// TIA Portal project "Project2" (V17)
// physical plc demo

(* hardware
DEVICE "S7-1500/ET200MP station_1"  S7-1500 station
   slot 0: "Rail_0"  Rack  6ES7 590-1***0-0AA0
   slot 1: "PLC_1"  CPU 1511-1 PN  6ES7 511-1AK02-0AB0  V2.9
      slot 3: "CPU display_1"  6ES7591-1AA00-0AA0
      slot 32768: "PROFINET interface_1"  X1
         slot 32769: "Port_1"  X1 P1
         slot 32770: "Port_2"  X1 P2
      slot 34817: "Virtual CP interface port_1"  Virtual CP interface port  Virtual CP interface port
DEVICE "HMI_1"  TP700 Comfort
   slot 0: "HMI_1"  TP700 Comfort  6AV2 124-0GC01-0AX0  17.0.0.0
   slot 1: "HMI_RT_1"  TP700 Comfort  6AV2 124-0GC01-0AX0  17.0.0.0
   slot 5: "HMI_1.IE_CP_1"  PROFINET Interface  17.0.0.0
      slot 1: "PROFINET Interface_1"  PROFINET Interface
         slot 1: "Port_1"  Port
         slot 2: "Port_2"  Port
   slot 7: "HMI_1.MPI/DP_CP_1"  MPI/DP Interface  17.0.0.0
DEVICE "ET 200SP station_1"  ET 200SP-Station
   slot 0: "RIO"  IM 155-6 PN/2 HF  6ES7 155-6AU01-0CN0  V4.2
   slot 0: "Rack_0"  Rack  6ES5 710-8MAx1
   slot 1: "DI 16x24VDC ST_1"  DI 16x24VDC ST  6ES7 131-6BH01-0BA0  V0.0
      slot 1: "DI 16x24VDC ST_1"  DI 16x24VDC ST
   slot 2: "DQ 16x24VDC/0.5A ST_1"  DQ 16x24VDC/0.5A ST  6ES7 132-6BH01-0BA0  V0.0
      slot 1: "DQ 16x24VDC/0.5A ST_1"  DQ 16x24VDC/0.5A ST
   slot 3: "AI 8xI 2-,4-wire BA_1"  AI 8xI 2-,4-wire BA  6ES7 134-6GF00-0AA1  V1.0
      slot 1: "AI 8xI 2-,4-wire BA_1"  AI 8xI 2-,4-wire BA
   slot 4: "AQ 4xU/I ST_1"  AQ 4xU/I ST  6ES7 135-6HD00-0BA1  V1.1
      slot 1: "AQ 4xU/I ST_1"  AQ 4xU/I ST
   slot 5: "Server module_1"  Server module  6ES7 193-6PA00-0AA0  V1.1
      slot 1: "Server module_1"  Server module
   slot 127: "BA 2xRJ45"  BA 2xRJ45  6ES7 193-6AR00-0AA0  V0.0
      slot 1: "Port_1"  X1 P1 R  6ES7 193-6AR00-0AA0  V0.0
      slot 2: "Port_2"  X1 P2 R  6ES7 193-6AR00-0AA0  V0.0
*)

// ===== PLC "PLC_1"  CPU 1511-1 PN =====

VAR_GLOBAL   // PLC tag table "Default tag table"
   "System_Byte" AT %MB1 : Byte;
   "FirstScan" AT %M1.0 : Bool;
   "DiagStatusUpdate" AT %M1.1 : Bool;
   "AlwaysTRUE" AT %M1.2 : Bool;
   "AlwaysFALSE" AT %M1.3 : Bool;
   "Clock_Byte" AT %MB0 : Byte;
   "Clock_10Hz" AT %M0.0 : Bool;
   "Clock_5Hz" AT %M0.1 : Bool;
   "Clock_2.5Hz" AT %M0.2 : Bool;
   "Clock_2Hz" AT %M0.3 : Bool;
   "Clock_1.25Hz" AT %M0.4 : Bool;
   "Clock_1Hz" AT %M0.5 : Bool;
   "Clock_0.625Hz" AT %M0.6 : Bool;
   "Clock_0.5Hz" AT %M0.7 : Bool;
   "Motor_Cikis" AT %QW2 : Int;
   "Motor_Ariza" AT %I0.0 : Bool;
END_VAR

DATA_BLOCK "Program_parameters_DB"   // DB1
{ S7_Optimized_Access := 'TRUE' }
VERSION : 0.1
   VAR
      QMotor1_Start : Bool;
      QMotor2_Start : Bool;
      QMotor3_Start : Bool;
      IMotor1_Fault : Bool;
      IMotor2_Fault : Bool;
      IMotor3_Fault : Bool;
      AQMotor1_Freq : Int;
      AQMotor2_Freq : Int;
      AQMotor3_Freq : Int;
   END_VAR
BEGIN
END_DATA_BLOCK

DATA_BLOCK "HMI_parameters_DB"   // DB2
{ S7_Optimized_Access := 'TRUE' }
VERSION : 0.1
   VAR
      HMI_Mode_Auto : Bool;
      HMI_M1_Manual_Start : Bool;
      HMI_M2_Manual_Start : Bool;
      HMI_M3_Manual_Start : Bool;
      HMI_M1_Manual_Speed : Real;
      HMI_M2_Manual_Speed : Real;
      HMI_M3_Manual_Speed : Real;
      HMI_M1_Running : Bool;
      HMI_M2_Running : Bool;
      HMI_M3_Running : Bool;
      HMI_M1_Fault : Bool;
      HMI_M2_Fault : Bool;
      HMI_M3_Fault : Bool;
   END_VAR
BEGIN
END_DATA_BLOCK

DATA_BLOCK "FB_Motor3_Sürücü_DB"   // DB3
{ S7_Optimized_Access := 'TRUE' }
VERSION : 0.1
// stored: InstanceOfName FB_Motor_Sürücü
"FB_Motor_Sürücü"
BEGIN
END_DATA_BLOCK

DATA_BLOCK "Data_block_1"   // DB4
{ S7_Optimized_Access := 'TRUE' }
VERSION : 0.1
   VAR
      man : Bool;
      Alarm : Int;
   END_VAR
BEGIN
END_DATA_BLOCK

DATA_BLOCK "FB_Motor1_Sürücü_DB"   // DB6
{ S7_Optimized_Access := 'TRUE' }
VERSION : 0.1
// stored: InstanceOfName FB_Motor_Sürücü
"FB_Motor_Sürücü"
BEGIN
END_DATA_BLOCK

DATA_BLOCK "FB_Motor2_Sürücü_DB"   // DB7
{ S7_Optimized_Access := 'TRUE' }
VERSION : 0.1
// stored: InstanceOfName FB_Motor_Sürücü
"FB_Motor_Sürücü"
BEGIN
END_DATA_BLOCK

FUNCTION_BLOCK "FB_Motor_Sürücü"   // FB1, LAD
{ S7_Optimized_Access := 'TRUE' }
VERSION : 0.1
   VAR_INPUT
      Enable : Bool;
      Mo_Auto : Bool;
      Man_Start : Bool;
      Man_Speed_Hz : Real;
      Driver_Fault : Bool;
   END_VAR
   VAR_OUTPUT
      Start_Out : Bool;
      Analog_Out : Int;
      Running : Bool;
      Alarm : Bool;
   END_VAR
   VAR_TEMP
      Target_Hz : Real;
      Norm_Val : Real;
   END_VAR
BEGIN

REGION Network 1
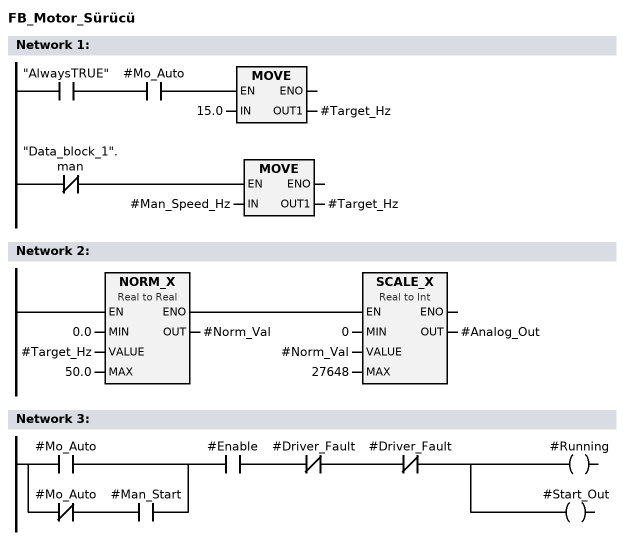
   RUNG wire#powerrail
      Contact( "AlwaysTRUE" )
      Contact( #Mo_Auto )
      Move(in := 15.0, out1 => #Target_Hz)
   END_RUNG
   RUNG wire#powerrail
      I_Contact( "Data_block_1".man )
      Move(in := #Man_Speed_Hz, out1 => #Target_Hz)
   END_RUNG
   // the same network as SCL:
   IF "AlwaysTRUE" AND #Mo_Auto THEN #Target_Hz := 15.0; END_IF;
   IF NOT "Data_block_1".man THEN #Target_Hz := #Man_Speed_Hz; END_IF;
END_REGION

REGION Network 2
   RUNG wire#powerrail
      { S7_Templates := "[SrcType := Real, DestType := Real]" } Normalize(min := 0.0, value := #Target_Hz, max := 50.0, out => #Norm_Val)
      { S7_Templates := "[SrcType := Real, DestType := Int]" } Scale(min := 0, value := #Norm_Val, max := 27648, out => #Analog_Out)
   END_RUNG
   // the same network as SCL:
   #Norm_Val := NORM_X(MIN := 0.0, VALUE := #Target_Hz, MAX := 50.0);
   #Analog_Out := SCALE_X(MIN := 0, VALUE := #Norm_Val, MAX := 27648);
END_REGION

REGION Network 3
   RUNG wire#powerrail
      Contact( #Mo_Auto )
      wire#w1
      Contact( #Enable )
      I_Contact( #Driver_Fault )
      I_Contact( #Driver_Fault )
      wire#w2
      Coil( #Running )
   END_RUNG
   RUNG wire#powerrail
      I_Contact( #Mo_Auto )
      Contact( #Man_Start )
   END_RUNG wire#w1
   RUNG wire#w2
      Coil( #Start_Out )
   END_RUNG
   // the same network as SCL:
   #Running := (#Mo_Auto OR (NOT #Mo_Auto AND #Man_Start)) AND #Enable AND NOT #Driver_Fault AND NOT #Driver_Fault;
   #Start_Out := #Running;
END_REGION
END_FUNCTION_BLOCK

FUNCTION "FC_Example" : Void   // FC1, LAD
{ S7_Optimized_Access := 'TRUE' }
VERSION : 0.1
BEGIN
END_FUNCTION

ORGANIZATION_BLOCK "Main"   // OB1, LAD, ProgramCycle
TITLE = "Main Program Sweep (Cycle)"
{ S7_Optimized_Access := 'TRUE' }
VERSION : 0.1
   VAR_INPUT
      Initial_Call : Bool;   // Initial call of this OB
      Remanence : Bool;   // =True, if remanent data are available
   END_VAR
BEGIN

REGION Network 1
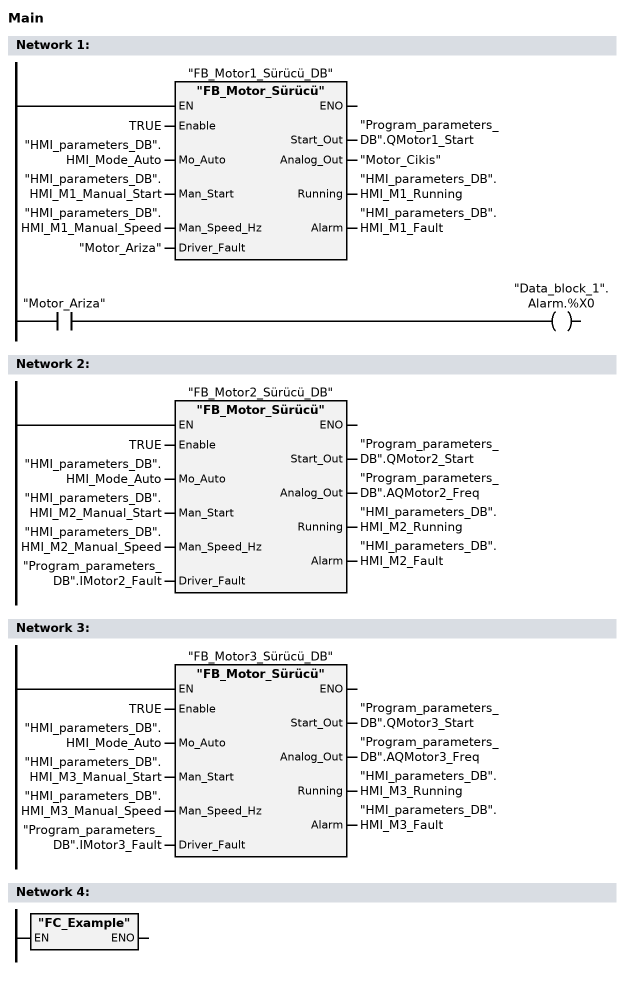
   RUNG wire#powerrail
      "FB_Motor1_Sürücü_DB"(Enable := TRUE, Mo_Auto := "HMI_parameters_DB".HMI_Mode_Auto, Man_Start := "HMI_parameters_DB".HMI_M1_Manual_Start, Man_Speed_Hz := "HMI_parameters_DB".HMI_M1_Manual_Speed, Driver_Fault := "Motor_Ariza", Start_Out => "Program_parameters_DB".QMotor1_Start, Analog_Out => "Motor_Cikis", Running => "HMI_parameters_DB".HMI_M1_Running, Alarm => "HMI_parameters_DB".HMI_M1_Fault)
   END_RUNG
   RUNG wire#powerrail
      Contact( "Motor_Ariza" )
      Coil( "Data_block_1".Alarm.%X0 )
   END_RUNG
   // the same network as SCL:
   "FB_Motor1_Sürücü_DB"(Enable := TRUE,   // "FB_Motor_Sürücü"
                         Mo_Auto := "HMI_parameters_DB".HMI_Mode_Auto,
                         Man_Start := "HMI_parameters_DB".HMI_M1_Manual_Start,
                         Man_Speed_Hz := "HMI_parameters_DB".HMI_M1_Manual_Speed,
                         Driver_Fault := "Motor_Ariza",
                         Start_Out => "Program_parameters_DB".QMotor1_Start,
                         Analog_Out => "Motor_Cikis",
                         Running => "HMI_parameters_DB".HMI_M1_Running,
                         Alarm => "HMI_parameters_DB".HMI_M1_Fault);
   "Data_block_1".Alarm.%X0 := "Motor_Ariza";
END_REGION

REGION Network 2
   RUNG wire#powerrail
      "FB_Motor2_Sürücü_DB"(Enable := TRUE, Mo_Auto := "HMI_parameters_DB".HMI_Mode_Auto, Man_Start := "HMI_parameters_DB".HMI_M2_Manual_Start, Man_Speed_Hz := "HMI_parameters_DB".HMI_M2_Manual_Speed, Driver_Fault := "Program_parameters_DB".IMotor2_Fault, Start_Out => "Program_parameters_DB".QMotor2_Start, Analog_Out => "Program_parameters_DB".AQMotor2_Freq, Running => "HMI_parameters_DB".HMI_M2_Running, Alarm => "HMI_parameters_DB".HMI_M2_Fault)
   END_RUNG
   // the same network as SCL:
   "FB_Motor2_Sürücü_DB"(Enable := TRUE,   // "FB_Motor_Sürücü"
                         Mo_Auto := "HMI_parameters_DB".HMI_Mode_Auto,
                         Man_Start := "HMI_parameters_DB".HMI_M2_Manual_Start,
                         Man_Speed_Hz := "HMI_parameters_DB".HMI_M2_Manual_Speed,
                         Driver_Fault := "Program_parameters_DB".IMotor2_Fault,
                         Start_Out => "Program_parameters_DB".QMotor2_Start,
                         Analog_Out => "Program_parameters_DB".AQMotor2_Freq,
                         Running => "HMI_parameters_DB".HMI_M2_Running,
                         Alarm => "HMI_parameters_DB".HMI_M2_Fault);
END_REGION

REGION Network 3
   RUNG wire#powerrail
      "FB_Motor3_Sürücü_DB"(Enable := TRUE, Mo_Auto := "HMI_parameters_DB".HMI_Mode_Auto, Man_Start := "HMI_parameters_DB".HMI_M3_Manual_Start, Man_Speed_Hz := "HMI_parameters_DB".HMI_M3_Manual_Speed, Driver_Fault := "Program_parameters_DB".IMotor3_Fault, Start_Out => "Program_parameters_DB".QMotor3_Start, Analog_Out => "Program_parameters_DB".AQMotor3_Freq, Running => "HMI_parameters_DB".HMI_M3_Running, Alarm => "HMI_parameters_DB".HMI_M3_Fault)
   END_RUNG
   // the same network as SCL:
   "FB_Motor3_Sürücü_DB"(Enable := TRUE,   // "FB_Motor_Sürücü"
                         Mo_Auto := "HMI_parameters_DB".HMI_Mode_Auto,
                         Man_Start := "HMI_parameters_DB".HMI_M3_Manual_Start,
                         Man_Speed_Hz := "HMI_parameters_DB".HMI_M3_Manual_Speed,
                         Driver_Fault := "Program_parameters_DB".IMotor3_Fault,
                         Start_Out => "Program_parameters_DB".QMotor3_Start,
                         Analog_Out => "Program_parameters_DB".AQMotor3_Freq,
                         Running => "HMI_parameters_DB".HMI_M3_Running,
                         Alarm => "HMI_parameters_DB".HMI_M3_Fault);
END_REGION

REGION Network 4
   RUNG wire#powerrail
      "FC_Example"()
   END_RUNG
   // the same network as SCL:
   "FC_Example"();
END_REGION
END_ORGANIZATION_BLOCK

(* ===== HMI "HMI_RT_1" =====
system functions are stored by id; their names below are inferred from use
connection "HMI_Connection_1": ETHERNET, S7_1500_OMS

HMI tags "Default tag table"
   "Tag_ScreenNumber" : UInt, internal
   "Data_block_1_Alarm" : Int = PLC Data_block_1.Alarm, 1 s
   "HMI_parameters_DB_HMI_Mode_Auto" : Bool = PLC HMI_parameters_DB.HMI_Mode_Auto, 1 s
   "HMI_parameters_DB_HMI_M1_Running" : Bool = PLC HMI_parameters_DB.HMI_M1_Running, 1 s
   "HMI_parameters_DB_HMI_M2_Running" : Bool = PLC HMI_parameters_DB.HMI_M2_Running, 1 s
   "HMI_parameters_DB_HMI_M3_Running" : Bool = PLC HMI_parameters_DB.HMI_M3_Running, 1 s
   "HMI_parameters_DB_HMI_M1_Manual_Start" : Bool = PLC HMI_parameters_DB.HMI_M1_Manual_Start, 1 s
   "HMI_parameters_DB_HMI_M2_Manual_Start" : Bool = PLC HMI_parameters_DB.HMI_M2_Manual_Start, 1 s
   "HMI_parameters_DB_HMI_M3_Manual_Start" : Bool = PLC HMI_parameters_DB.HMI_M3_Manual_Start, 1 s
   "HMI_parameters_DB_HMI_M1_Manual_Speed" : Real = PLC HMI_parameters_DB.HMI_M1_Manual_Speed, 1 s
   "HMI_parameters_DB_HMI_M2_Manual_Speed" : Real = PLC HMI_parameters_DB.HMI_M2_Manual_Speed, 1 s
   "HMI_parameters_DB_HMI_M3_Manual_Speed" : Real = PLC HMI_parameters_DB.HMI_M3_Manual_Speed, 1 s
   "HMI_parameters_DB_HMI_M1_Fault" : Bool = PLC HMI_parameters_DB.HMI_M1_Fault, 1 s
   "HMI_parameters_DB_HMI_M2_Fault" : Bool = PLC HMI_parameters_DB.HMI_M2_Fault, 1 s
   "HMI_parameters_DB_HMI_M3_Fault" : Bool = PLC HMI_parameters_DB.HMI_M3_Fault, 1 s

discrete alarms
   1: 'First Motor Driver Fault!', class Errors, trigger "HMI_parameters_DB_HMI_M1_Fault" bit 0

Template "Template_1" 800x420
   Button "Exit" at 720,360 size 78x58; TextOff 'Exit'; PictureOff "ExitRuntime_TP700_Comfort_TR"; PictureOn "ExitRuntime_TP700_Comfort_TR"
      on Release: StopRuntime(0)
   Button "Template_Button" at 640,360 size 78x58; TextOff 'Text'
   Button "Template_Button_1" at 560,360 size 78x58; TextOff 'Text'
   Button "Template_Button_2" at 480,360 size 78x58; TextOff 'Text'
   Button "Template_Button_3" at 400,360 size 78x58; TextOff 'Text'
   Button "Template_Button_4" at 321,360 size 78x58; TextOff 'Text'
   Button "Template_Button_5" at 241,360 size 78x58; TextOff 'Text'
   Button "Template_Button_6" at 161,360 size 78x58; TextOff 'Text'
   Button "Alarms" at 81,360 size 78x58; TextOff 'Alarms'; PictureOff "AlarmDisplay_TP700_Comfort_TR"; PictureOn "AlarmDisplay_TP700_Comfort_TR"
      on Release: function_ef3f5d25("Alarm window_Unacknowledged", -1)
   Button "Start screen" at 1,360 size 78x58; TextOff 'Start screen'; PictureOff "NavigateHome_TP700_Comfort_TR"; PictureOn "NavigateHome_TP700_Comfort_TR"
      on Release: ActivateScreen("Root screen", 0)

screen "Screen_1" 800x420
   Switch "Switch_1" at 14,4 size 120x88; CaptionText 'Switch'; TextOff 'MANUAL'; TextOn 'OTOMATIC (15 Hz)'
      ProcessValue <- "HMI_parameters_DB_HMI_Mode_Auto"
   GraphicView "Graphic view_1" at 175,69 size 186x82; Picture "Graphic_8"
      Appearance <- "HMI_parameters_DB_HMI_M1_Running"
   Button "Button_1" at 180,19 size 96x32; TextOff 'M1_START'
      on Press: function_b14e0dd5("HMI_parameters_DB_HMI_M1_Manual_Start", 0)
   Button "Button_2" at 396,16 size 96x32; TextOff 'M2_START'
      on Press: function_b14e0dd5("HMI_parameters_DB_HMI_M2_Manual_Start", 0)
   GraphicView "Graphic view_2" at 381,55 size 187x105; Picture "Graphic_11"
      Appearance <- "HMI_parameters_DB_HMI_M2_Running"
   GraphicView "Graphic view_3" at 613,55 size 187x105; Picture "Graphic_12"
      Appearance <- "HMI_parameters_DB_HMI_M3_Running"
   Button "Button_3" at 623,20 size 96x32; TextOff 'M3_START'
      on Press: function_b14e0dd5("HMI_parameters_DB_HMI_M3_Manual_Start", 0)
   IOField "I/O field_1" at 180,169 size 96x32; FormatPattern 999.99
      ProcessValue <- "HMI_parameters_DB_HMI_M1_Manual_Speed"
   IOField "I/O field_2" at 381,169 size 96x32; FormatPattern 999.99
      ProcessValue <- "HMI_parameters_DB_HMI_M2_Manual_Speed"
   IOField "I/O field_3" at 613,169 size 96x32; FormatPattern 999.99
      ProcessValue <- "HMI_parameters_DB_HMI_M3_Manual_Speed"
   Circle "Circle_1" at 203,258 size 48x48
      Appearance <- "HMI_parameters_DB_HMI_M1_Fault"
   Circle "Circle_2" at 406,251 size 48x48
      Appearance <- "HMI_parameters_DB_HMI_M2_Fault"
   Circle "Circle_3" at 636,251 size 48x48
      Appearance <- "HMI_parameters_DB_HMI_M3_Fault"
   TextField "Text field_1" at 204,226 size 88x23; Text 'M1_Fault'
   TextField "Text field_2" at 406,226 size 88x23; Text 'M2_Fault'
   TextField "Text field_3" at 635,226 size 88x23; Text 'M3_Fault'
   GraphicView "Graphic view_4" at 20,333 size 51x51; Picture "Graphic_1"
      Appearance <- "HMI_parameters_DB_HMI_M1_Fault"
*)